Yaskawa INFORM job: TCP_SHORT_SPIKE2.JBI

/JOB
//NAME TCP_SHORT_SPIKE2
///FOLDERNAME INNE
//POS
///NPOS 15,15,0,0,0,0
///TOOL 0
///POSTYPE PULSE
///PULSE
C00000=-4388,6378,88847,4334,105520,40804
C00001=51855,-19719,54378,3657,103962,51202
C00002=123924,-21071,53528,4017,103771,51322
C00003=161056,-23985,50068,4857,105083,41574
C00004=219900,-23897,50071,5782,105060,41912
C00005=-233447,-6475,72717,6132,105630,44357
C00006=-151980,-955,79142,6024,104420,50961
C00007=-123017,-3096,75835,6086,106531,39573
C00008=-41274,-13321,61783,-4327,108532,-25935
C00009=-60388,-51966,15809,-4514,98318,-36157
C00010=-171065,-40121,29466,-3475,101519,-41265
C00011=-222296,-74556,-3638,-641,91470,-10047
C00012=-32978,-102600,-22108,4632,68437,32093
C00013=35867,-72021,-2211,2906,85643,58705
C00014=-5467,-47820,20343,4238,99634,38748
BC00000=234605,127399,695029
BC00001=234605,127399,695029
BC00002=234605,127399,695029
BC00003=234605,127399,695029
BC00004=234605,127399,695029
BC00005=234605,127399,695029
BC00006=234605,127399,695029
BC00007=234605,127399,695029
BC00008=234605,127399,695029
BC00009=234605,127399,695029
BC00010=234605,127399,695029
BC00011=234605,127399,695029
BC00012=234605,127399,695029
BC00013=234605,127399,695027
BC00014=234605,127399,695029
//INST
///DATE 2023/10/04 15:16
///ATTR SC,RW
///GROUP1 RB1,BS1
NOP
MOVJ C00000 BC00000 VJ=0.78
MOVJ C00001 BC00001 VJ=0.78
MOVJ C00002 BC00002 VJ=0.78
MOVJ C00003 BC00003 VJ=0.78
MOVJ C00004 BC00004 VJ=0.78
MOVJ C00005 BC00005 VJ=0.78
MOVJ C00006 BC00006 VJ=0.78
MOVJ C00007 BC00007 VJ=0.78
MOVJ C00008 BC00008 VJ=0.78
MOVJ C00009 BC00009 VJ=0.78
MOVJ C00010 BC00010 VJ=0.78
MOVJ C00011 BC00011 VJ=0.78
MOVJ C00012 BC00012 VJ=0.78
MOVJ C00013 BC00013 VJ=0.78
MOVJ C00014 BC00014 VJ=0.78
END
